# EPICS substitutions: PIP-II/RFPI2/rfpi-fdr-sw-main-ioc/kriaApp/Db/expert.substitutions
file expert.template {
pattern{ acc, sys, group, num, cav }
{ PIP2IT, pHB650, RFPI, zynq, C1 }
{ PIP2IT, pHB650, RFPI, zynq, C2 }
{ PIP2IT, pHB650, RFPI, zynq, C3 }
{ PIP2IT, pHB650, RFPI, zynq, C4 }
}
